// TIA Portal V19 export
// export: Created 2018-02-02T09:20:05.7051255Z, ExportSetting None, DisplayName Totally Integrated Automation Portal, DisplayVersion V19, DisplayName TIA Portal Openness, DisplayVersion V19, DisplayName SINAMICS Startdrive, DisplayVersion V19, DisplayName STEP 7 Professional, DisplayVersion V19, DisplayName STEP 7 Safety, DisplayVersion V19, DisplayName WinCC Professional, DisplayVersion V19, DisplayName SIMATIC Visualization Architect, DisplayVersion V19
FUNCTION_BLOCK ""   // FB, GRAPH
{ S7_Optimized_Access := 'TRUE' }
// stored: InitialValuesAcquisition false, SetENOAutomatically false
   // inherited from GRAPH_BASE
   VAR_INPUT
      OFF_SQ { ExternalAccessible := 'False'; ExternalVisible := 'False'; ExternalWritable := 'False'} : Bool := false;   // Kette ausschalten
      INIT_SQ { ExternalAccessible := 'False'; ExternalVisible := 'False'; ExternalWritable := 'False'} : Bool := false;   // Kette in Initialzustand versetzen
      ACK_EF { ExternalAccessible := 'False'; ExternalVisible := 'False'; ExternalWritable := 'False'} : Bool := false;   // Alle Fehler und Störungen quittieren
      S_PREV { ExternalAccessible := 'False'; ExternalVisible := 'False'; ExternalWritable := 'False'} : Bool := false;   // Vorherigen Schritt am Parameter S_NO ausgeben
      S_NEXT { ExternalAccessible := 'False'; ExternalVisible := 'False'; ExternalWritable := 'False'} : Bool := false;   // Nächsten Schritt am Parameter S_NO anzeigen
      SW_AUTO { ExternalAccessible := 'False'; ExternalVisible := 'False'; ExternalWritable := 'False'} : Bool := false;   // Automatischer Betrieb
      SW_TAP { ExternalAccessible := 'False'; ExternalVisible := 'False'; ExternalWritable := 'False'} : Bool := false;   // Halbautomatisch/Weiterschalten mit Transition
      SW_TOP { ExternalAccessible := 'False'; ExternalVisible := 'False'; ExternalWritable := 'False'} : Bool := false;   // Halbautomatisch/Ignoriere Transition
      SW_MAN { ExternalAccessible := 'False'; ExternalVisible := 'False'; ExternalWritable := 'False'} : Bool := false;   // Handbetrieb
      S_SEL { ExternalAccessible := 'False'; ExternalVisible := 'False'; ExternalWritable := 'False'} : Int := 0;   // Schritt auswählen, der an S_NO ausgegeben werden soll
      S_ON { ExternalAccessible := 'False'; ExternalVisible := 'False'; ExternalWritable := 'False'} : Bool := false;   // Schritt aktivieren, der an Parameter S_NO anliegt
      S_OFF { ExternalAccessible := 'False'; ExternalVisible := 'False'; ExternalWritable := 'False'} : Bool := false;   // Schritt deaktivieren, der an Parameter S_NO anliegt
      T_PUSH { ExternalAccessible := 'False'; ExternalVisible := 'False'; ExternalWritable := 'False'} : Bool := false;   // Schaltfreigabe für Transition im halbautomatischen Betrieb
   END_VAR
   VAR_OUTPUT
      S_NO { ExternalAccessible := 'False'; ExternalVisible := 'False'; ExternalWritable := 'False'} : Int := 0;   // Schrittnummer
      S_MORE { ExternalAccessible := 'False'; ExternalVisible := 'False'; ExternalWritable := 'False'} : Bool := false;   // Weitere Schritte sind vorhanden und können in S_NO angezeigt werden.
      S_ACTIVE { ExternalAccessible := 'False'; ExternalVisible := 'False'; ExternalWritable := 'False'} : Bool := false;   // Schritt, der an Parameter S_NO angezeigt wird, ist aktiv
      ERR_FLT { ExternalAccessible := 'False'; ExternalVisible := 'False'; ExternalWritable := 'False'} : Bool := false;   // Sammelfehler Interlock oder Supervision
      AUTO_ON { ExternalAccessible := 'False'; ExternalVisible := 'False'; ExternalWritable := 'False'} : Bool := false;   // Automatischer Betrieb eingeschaltet
      TAP_ON { ExternalAccessible := 'False'; ExternalVisible := 'False'; ExternalWritable := 'False'} : Bool := false;   // Halbautomatischer Betrieb/Schritt mit Transition eingeschaltet
      TOP_ON { ExternalAccessible := 'False'; ExternalVisible := 'False'; ExternalWritable := 'False'} : Bool := false;   // Halbautomatischer Betrieb/Ignoriere Transition eingeschaltet
      MAN_ON { ExternalAccessible := 'False'; ExternalVisible := 'False'; ExternalWritable := 'False'} : Bool := false;   // Handbetrieb eingeschaltet
   END_VAR
BEGIN
   // sequencer 1: My step sequence
   // My step sequecne comment
END_FUNCTION_BLOCK
